PROGRAM PRG_ManualControl
VAR
	
	rMotorsActualPosition : ARRAY[1..3] OF LREAL;
	rValvesActualPosition : ARRAY[1..5] OF LREAL;
	rPumpsActualPosition  : ARRAY[1..10] OF LREAL;
	rDegreesPerVolume 	  : ARRAY[1..10] OF LREAL;
	
	aPumpsActivated		  : ARRAY[1..10] OF BOOL;
	aPumpsDirection		  : ARRAY[1..10] OF E_PumpDirection;
	aPumpsSpeed			  : ARRAY[1..10] OF REAL;
	aPumpsVolume		  : ARRAY[1..10] OF REAL;
	aPumpsDistance		  : ARRAY[1..10] OF UINT;
	bRunPumpsBySpeed	  : BOOL := FALSE;
	bRunPumpsByVolume	  : BOOL := FALSE;
	bRunPumpsByDistance	  : BOOL := FALSE;
	
	aMotorBusy	: ARRAY[1..3] OF BOOL;
	
	fbPumpsController : FB_AllPumpsController;

	i : INT; 
	
	//interlock Variables
	iTargetPosM2 : INT;
    rActualPosM3 : LREAL;
    rTol         : LREAL := 3.0; // tolerância para considerar posição "alinhada"
    bAllowMoveM2 : BOOL := TRUE;
		
END_VAR

//Motors Manual jog handling 
MotorsJog();
MotorsActualPosition();

//New Manual Screen commands test area ##########################################################
(* <Motors> -----------------------------------------------------------------------------------------------------------------------------------------------------------------------------------*)

(*<M1 Motor>*)
//Move M1 by HMI combobox manual mode
IF GVL_HMI.aManualMotorsCmd[1].bRun THEN
	GVL_HMI.aManualMotorsCmd[1].bRun := NOT GVL_Motion.aMotors[1].MoveAbsolute(	rPosition := GVL_Settings.stMachineParam.aM1Position[GVL_HMI.aManualMotorsCmd[1].iPosition],
                        														rVelocity := GVL_Settings.stMachineParam.rM1Velocity,
                        														rAcc := GVL_Settings.stMachineParam.rM1Accleration,
                       															rDec := GVL_Settings.stMachineParam.rM1Deceleration
																				);
END_IF
//Stop Moviment M1 by HMI manual mode button
IF GVL_HMI.aManualMotorsCmd[1].bStop THEN
	GVL_HMI.aManualMotorsCmd[1].bStop := NOT GVL_Motion.aMotors[1].Stop();
END_IF
(*<\M1 Motor>*)

(*<M2 Motor>*)
//Move M2 by HMI combobox manual mode
iTargetPosM2 := GVL_HMI.aManualMotorsCmd[2].iPosition;
rActualPosM3 := rMotorsActualPosition[3];

//Interlock move for M2 base on M3 position
CASE iTargetPosM2 OF
    3: // Fill Vials
        bAllowMoveM2 := (
            ABS(rActualPosM3 - GVL_Settings.stMachineParam.aM3Position[2]) <= rTol OR
            ABS(rActualPosM3 - GVL_Settings.stMachineParam.aM3Position[3]) <= rTol OR
            ABS(rActualPosM3 - GVL_Settings.stMachineParam.aM3Position[4]) <= rTol OR
            ABS(rActualPosM3 - GVL_Settings.stMachineParam.aM3Position[5]) <= rTol
        );

    4: // Calibration
        bAllowMoveM2 := ABS(rActualPosM3 - GVL_Settings.stMachineParam.aM3Position[6]) <= rTol;

    ELSE
        bAllowMoveM2 := TRUE;
END_CASE

//M2 Moviment if there is no interlock
IF GVL_HMI.aManualMotorsCmd[2].bRun THEN
    IF bAllowMoveM2 THEN
        GVL_HMI.aManualMotorsCmd[2].bRun := NOT GVL_Motion.aMotors[2].MoveAbsolute(
            rPosition := GVL_Settings.stMachineParam.aM2Position[iTargetPosM2],
            rVelocity := GVL_Settings.stMachineParam.rM2Velocity,
            rAcc := GVL_Settings.stMachineParam.rM2Accleration,
            rDec := GVL_Settings.stMachineParam.rM2Deceleration
        );
    ELSE
        GVL_HMI.aManualMotorsCmd[2].bRun := FALSE;
        // TODO: Block flag or alarm
    END_IF
END_IF

//Stop Moviment M2 by HMI manual mode button
IF GVL_HMI.aManualMotorsCmd[2].bStop THEN
	GVL_HMI.aManualMotorsCmd[2].bStop := NOT GVL_Motion.aMotors[2].Stop();
END_IF
(*<\M2 Motor>*)

(*<M3 Motor>*)
//Interlock by M2 Position
IF GVL_HMI.aManualMotorsCmd[3].bRun THEN
    IF ABS(rMotorsActualPosition[2] - GVL_Settings.stMachineParam.aM2Position[1]) > rTol THEN
        //If M2 it is not in Home Position, M3 move cannot be done
        GVL_HMI.aManualMotorsCmd[3].bRun := FALSE;
        // TODO: Block flag or alarm
    ELSE
        GVL_HMI.aManualMotorsCmd[3].bRun := NOT GVL_Motion.aMotors[3].MoveAbsolute(
            rPosition := GVL_Settings.stMachineParam.aM3Position[GVL_HMI.aManualMotorsCmd[3].iPosition],
            rVelocity := GVL_Settings.stMachineParam.rM3Velocity,
            rAcc := GVL_Settings.stMachineParam.rM3Accleration,
            rDec := GVL_Settings.stMachineParam.rM3Deceleration
        );
    END_IF
END_IF
//Stop Moviment M2 by HMI manual mode button
IF GVL_HMI.aManualMotorsCmd[3].bStop THEN
	GVL_HMI.aManualMotorsCmd[3].bStop := NOT GVL_Motion.aMotors[3].Stop();
END_IF
(*<\M3 Motor>*)

(* <Valves> -----------------------------------------------------------------------------------------------------------------------------------------------------------------------------------*)

(*<Valve 1>*)
//Move Valve 1 by HMI combobox manual mode
IF GVL_HMI.aManualValvesCmd[1].bMove THEN
	GVL_HMI.aManualValvesCmd[1].bMove := NOT GVL_Motion.aValvesObj[1].MoveValve( iPosition := GVL_HMI.aManualValvesCmd[1].iTargetPos ,rVelocity := 1500, rAcc := 1000, rDec := 1000);
END_IF

//Stop Moviment Valve 1 by HMI manual mode button
IF GVL_HMI.aManualValvesCmd[1].bStop THEN
	GVL_HMI.aManualValvesCmd[1].bStop := NOT GVL_Motion.aValvesObj[1].Stop();
END_IF
(*<\Valve 1>*)

(*<Valve 2>*)
//Move Valve 2 by HMI combobox manual mode
IF GVL_HMI.aManualValvesCmd[2].bMove THEN
	GVL_HMI.aManualValvesCmd[2].bMove := NOT GVL_Motion.aValvesObj[2].MoveValve( iPosition := GVL_HMI.aManualValvesCmd[2].iTargetPos ,rVelocity := 1500, rAcc := 1000, rDec := 1000);
END_IF

//Stop Moviment Valve 2 by HMI manual mode button
IF GVL_HMI.aManualValvesCmd[2].bStop THEN
	GVL_HMI.aManualValvesCmd[2].bStop := NOT GVL_Motion.aValvesObj[2].Stop();
END_IF
(*<\Valve 2>*)

(*<Valve 3>*)
//Move Valve 3 by HMI combobox manual mode
IF GVL_HMI.aManualValvesCmd[3].bMove THEN
	GVL_HMI.aManualValvesCmd[3].bMove := NOT GVL_Motion.aValvesObj[3].MoveValve( iPosition := GVL_HMI.aManualValvesCmd[3].iTargetPos ,rVelocity := 1500, rAcc := 1000, rDec := 1000);
END_IF

//Stop Moviment Valve 3 by HMI manual mode button
IF GVL_HMI.aManualValvesCmd[3].bStop THEN
	GVL_HMI.aManualValvesCmd[3].bStop := NOT GVL_Motion.aValvesObj[3].Stop();
END_IF
(*<\Valve 3>*)

(*<Valve 4>*)
//Move Valve 4 by HMI combobox manual mode
IF GVL_HMI.aManualValvesCmd[4].bMove THEN
	GVL_HMI.aManualValvesCmd[4].bMove := NOT GVL_Motion.aValvesObj[4].MoveValve( iPosition := GVL_HMI.aManualValvesCmd[4].iTargetPos ,rVelocity := 1500, rAcc := 1000, rDec := 1000);
END_IF

//Stop Moviment Valve 4 by HMI manual mode button
IF GVL_HMI.aManualValvesCmd[4].bStop THEN
	GVL_HMI.aManualValvesCmd[4].bStop := NOT GVL_Motion.aValvesObj[4].Stop();
END_IF
(*<\Valve 4>*)

(*<Valve 5>*)
//Move Valve 5 by HMI combobox manual mode
IF GVL_HMI.aManualValvesCmd[5].bMove THEN
	GVL_HMI.aManualValvesCmd[5].bMove := NOT GVL_Motion.aValvesObj[5].MoveValve( iPosition := GVL_HMI.aManualValvesCmd[5].iTargetPos ,rVelocity := 1500, rAcc := 1000, rDec := 1000);
END_IF

//Stop Moviment Valve 5 by HMI manual mode button
IF GVL_HMI.aManualValvesCmd[5].bStop THEN
	GVL_HMI.aManualValvesCmd[5].bStop := NOT GVL_Motion.aValvesObj[5].Stop();
END_IF
(*<\Valve 5>*)

(* <Pumps> -----------------------------------------------------------------------------------------------------------------------------------------------------------------------------------*)
(*<Move by Speed>*)
IF GVL_HMI.bRunPumpsBySpeedBt THEN //Fill up the pump arrays and trigger pumps 
	FOR i := 1 TO 10 DO
		aPumpsActivated[i] := GVL_HMI.aManualPumpsCmd[i].bActive;
		aPumpsDirection[i] := GVL_HMI.aManualPumpsCmd[i].eDirection;
		aPumpsSpeed[i] := GVL_HMI.aManualPumpsCmd[i].rSpeed * 6;
	END_FOR
	bRunPumpsBySpeed := TRUE;
	GVL_HMI.bRunPumpsBySpeedBt := FALSE;
END_IF
IF bRunPumpsBySpeed THEN //pumps movement
	bRunPumpsBySpeed := NOT fbPumpsController.MoveBySpeed(aPumpIds := aPumpsActivated, aVelocity := aPumpsSpeed, aPumpDirection := aPumpsDirection);
END_IF
(*<\Move by Speed>*)

(*<Move by Volume>*)
IF GVL_HMI.bRunPumpsByVolumeBt THEN //Fill up the pump arrays and trigger pumps 
	FOR i := 1 TO 10 DO
		aPumpsActivated[i] := GVL_HMI.aManualPumpsCmd[i].bActive;
		aPumpsDirection[i] := GVL_HMI.aManualPumpsCmd[i].eDirection;
		aPumpsSpeed[i] := GVL_HMI.aManualPumpsCmd[i].rSpeed * 6;
		aPumpsVolume[i] := GVL_HMI.aManualPumpsCmd[i].rVolume;
	END_FOR
	bRunPumpsByVolume := TRUE;
	GVL_HMI.bRunPumpsByVolumeBt := FALSE;
END_IF
IF bRunPumpsByVolume THEN //pumps movement
	bRunPumpsByVolume := NOT fbPumpsController.MoveByVolume(aPumpIds := aPumpsActivated, aVolume := aPumpsVolume, aPumpDirection := aPumpsDirection, aVelocity := aPumpsSpeed);
END_IF
(*<\Move by Volume>*)

(*<Move by Distance>*)
IF GVL_HMI.bRunPumpsByDistanceBt THEN //Fill up the pump arrays and trigger pumps 
	FOR i := 1 TO 10 DO
		aPumpsActivated[i] := GVL_HMI.aManualPumpsCmd[i].bActive;
		aPumpsDirection[i] := GVL_HMI.aManualPumpsCmd[i].eDirection;
		aPumpsSpeed[i] := GVL_HMI.aManualPumpsCmd[i].rSpeed * 6;
		aPumpsDistance[i] := GVL_HMI.aManualPumpsCmd[i].iDistance;
	END_FOR
	bRunPumpsByDistance := TRUE;
	GVL_HMI.bRunPumpsByDistanceBt := FALSE;
END_IF
IF bRunPumpsByDistance THEN //pumps movement
	bRunPumpsByDistance := NOT fbPumpsController.MoveByDistance(aPumpIds := aPumpsActivated, aRevolutions := aPumpsDistance, aPumpDirection := aPumpsDirection, aVelocity := aPumpsSpeed);
END_IF
(*<\Move by Distance>*)

(*<Stop All Pumps>*)
IF GVL_HMI.bStopPumpsBt THEN
	GVL_HMI.bStopPumpsBt := NOT fbPumpsController.StopAllPumps();
END_IF
(*<\Stop All Pumps>*)

(* <\Pumps> ----------------------------------------------------------------------------------------------------------------------------------------------------------------------------------*)

ACTION MotorsActualPosition:
// Get Motors Actual Position
rMotorsActualPosition[1] := GVL_Motion.aMotors[1].GetPosition();
rMotorsActualPosition[2] := GVL_Motion.aMotors[2].GetPosition();
rMotorsActualPosition[3] := GVL_Motion.aMotors[3].GetPosition();
rValvesActualPosition[1] := GVL_Motion.aValvesObj[1].GetPosition();
rValvesActualPosition[2] := GVL_Motion.aValvesObj[2].GetPosition();
rValvesActualPosition[3] := GVL_Motion.aValvesObj[3].GetPosition();
rValvesActualPosition[4] := GVL_Motion.aValvesObj[4].GetPosition();
rValvesActualPosition[5] := GVL_Motion.aValvesObj[5].GetPosition();
rPumpsActualPosition[1] := GVL_Motion.aPumpsLinear[1].GetPosition();
rPumpsActualPosition[2] := GVL_Motion.aPumpsLinear[2].GetPosition();
rPumpsActualPosition[3] := GVL_Motion.aPumpsLinear[3].GetPosition();
rPumpsActualPosition[4] := GVL_Motion.aPumpsLinear[4].GetPosition();
rPumpsActualPosition[5] := GVL_Motion.aPumpsLinear[5].GetPosition();
rPumpsActualPosition[6] := GVL_Motion.aPumpsLinear[6].GetPosition();
rPumpsActualPosition[7] := GVL_Motion.aPumpsLinear[7].GetPosition();
rPumpsActualPosition[8] := GVL_Motion.aPumpsLinear[8].GetPosition();
rPumpsActualPosition[9] := GVL_Motion.aPumpsLinear[9].GetPosition();
rPumpsActualPosition[10] := GVL_Motion.aPumpsLinear[10].GetPosition();

//Linear Motors - M1, M2, M3
GVL_Motion.M1Motor.rActualPosition := F_ROUND_REAL(rInput := TO_REAL(rMotorsActualPosition[1]), iDecimalPlaces := 2)* -1;
GVL_Motion.M2Motor.rActualPosition := F_ROUND_REAL(rInput := TO_REAL(rMotorsActualPosition[2]), iDecimalPlaces := 2)* -1;
GVL_Motion.M3Motor.rActualPosition := F_ROUND_REAL(rInput := TO_REAL(rMotorsActualPosition[3]), iDecimalPlaces := 2)* -1;

//Vici Valves - M4 to M8
GVL_Motion.aValves[1].rActualPosition := F_ROUND_REAL(rInput := TO_REAL(rValvesActualPosition[1]), iDecimalPlaces := 2);
GVL_Motion.aValves[2].rActualPosition := F_ROUND_REAL(rInput := TO_REAL(rValvesActualPosition[2]), iDecimalPlaces := 2);
GVL_Motion.aValves[3].rActualPosition := F_ROUND_REAL(rInput := TO_REAL(rValvesActualPosition[3]), iDecimalPlaces := 2);
GVL_Motion.aValves[4].rActualPosition := F_ROUND_REAL(rInput := TO_REAL(rValvesActualPosition[4]), iDecimalPlaces := 2);
GVL_Motion.aValves[5].rActualPosition := F_ROUND_REAL(rInput := TO_REAL(rValvesActualPosition[5]), iDecimalPlaces := 2);

//Linear pumps - 1 to 10
GVL_Motion.aPumps[1].Linear.rActualPosition  := F_ROUND_REAL(rInput := TO_REAL(rPumpsActualPosition[1]), iDecimalPlaces := 2)* -1;
GVL_Motion.aPumps[2].Linear.rActualPosition  := F_ROUND_REAL(rInput := TO_REAL(rPumpsActualPosition[2]), iDecimalPlaces := 2)* -1;
GVL_Motion.aPumps[3].Linear.rActualPosition  := F_ROUND_REAL(rInput := TO_REAL(rPumpsActualPosition[3]), iDecimalPlaces := 2)* -1;
GVL_Motion.aPumps[4].Linear.rActualPosition  := F_ROUND_REAL(rInput := TO_REAL(rPumpsActualPosition[4]), iDecimalPlaces := 2)* -1;
GVL_Motion.aPumps[5].Linear.rActualPosition  := F_ROUND_REAL(rInput := TO_REAL(rPumpsActualPosition[5]), iDecimalPlaces := 2)* -1;
GVL_Motion.aPumps[6].Linear.rActualPosition  := F_ROUND_REAL(rInput := TO_REAL(rPumpsActualPosition[6]), iDecimalPlaces := 2)* -1;
GVL_Motion.aPumps[7].Linear.rActualPosition  := F_ROUND_REAL(rInput := TO_REAL(rPumpsActualPosition[7]), iDecimalPlaces := 2)* -1;
GVL_Motion.aPumps[8].Linear.rActualPosition  := F_ROUND_REAL(rInput := TO_REAL(rPumpsActualPosition[8]), iDecimalPlaces := 2)* -1;
GVL_Motion.aPumps[9].Linear.rActualPosition  := F_ROUND_REAL(rInput := TO_REAL(rPumpsActualPosition[9]), iDecimalPlaces := 2)* -1;
GVL_Motion.aPumps[10].Linear.rActualPosition := F_ROUND_REAL(rInput := TO_REAL(rPumpsActualPosition[10]), iDecimalPlaces := 2)* -1;
END_ACTION

ACTION MotorsJog:
//Manual Motors Moviment

//Manual Moviment motor 1 - Stage Collection Vertical Axis
GVL_Motion.aMotors[1].Jog(bFwd := GVL_HMI.ManualMov.bMotorsJogFwd[1], bBwd := GVL_HMI.ManualMov.bMotorsJogBwd[1]);
//Manual Moviment motor 2 - Sample Recovery Vertical Axis
GVL_Motion.aMotors[2].Jog(bFwd := GVL_HMI.ManualMov.bMotorsJogFwd[2], bBwd := GVL_HMI.ManualMov.bMotorsJogBwd[2]);
//Manual Moviment motor 3 - Sample Recovery Horizontal Axis
GVL_Motion.aMotors[3].Jog(bFwd := GVL_HMI.ManualMov.bMotorsJogFwd[3], bBwd := GVL_HMI.ManualMov.bMotorsJogBwd[3]);

//Manual Moviment M4 - Valve 1 
GVL_Motion.aValvesObj[1].Jog(bFwd := GVL_HMI.ManualMov.bValvesJogFwd[1], bBwd := GVL_HMI.ManualMov.bValvesJogBwd[1]);
//Manual Moviment M5 - Valve 2 
GVL_Motion.aValvesObj[2].Jog(bFwd := GVL_HMI.ManualMov.bValvesJogFwd[2], bBwd := GVL_HMI.ManualMov.bValvesJogBwd[2]);
//Manual Moviment M6 - Valve 3
GVL_Motion.aValvesObj[3].Jog(bFwd := GVL_HMI.ManualMov.bValvesJogFwd[3], bBwd := GVL_HMI.ManualMov.bValvesJogBwd[3]);
//Manual Moviment M7 - Valve 4
GVL_Motion.aValvesObj[4].Jog(bFwd := GVL_HMI.ManualMov.bValvesJogFwd[4], bBwd := GVL_HMI.ManualMov.bValvesJogBwd[4]);
//Manual Moviment M8 - Valve 5
GVL_Motion.aValvesObj[5].Jog(bFwd := GVL_HMI.ManualMov.bValvesJogFwd[5], bBwd := GVL_HMI.ManualMov.bValvesJogBwd[5]);

//Manual Moviment Pump 1 - Linear
GVL_Motion.aPumpsLinear[1].Jog(bFwd := GVL_HMI.ManualMov.bPumpsLinearJogFwd[1], bBwd := GVL_HMI.ManualMov.bPumpsLinearJogBwd[1]);
//Manual Moviment Pump 2 - Linear
GVL_Motion.aPumpsLinear[2].Jog(bFwd := GVL_HMI.ManualMov.bPumpsLinearJogFwd[2], bBwd := GVL_HMI.ManualMov.bPumpsLinearJogBwd[2]);
//Manual Moviment Pump 3 - Linear
GVL_Motion.aPumpsLinear[3].Jog(bFwd := GVL_HMI.ManualMov.bPumpsLinearJogFwd[3], bBwd := GVL_HMI.ManualMov.bPumpsLinearJogBwd[3]);
//Manual Moviment Pump 4 - Linear
GVL_Motion.aPumpsLinear[4].Jog(bFwd := GVL_HMI.ManualMov.bPumpsLinearJogFwd[4], bBwd := GVL_HMI.ManualMov.bPumpsLinearJogBwd[4]);
//Manual Moviment Pump 5 - Linear
GVL_Motion.aPumpsLinear[5].Jog(bFwd := GVL_HMI.ManualMov.bPumpsLinearJogFwd[5], bBwd := GVL_HMI.ManualMov.bPumpsLinearJogBwd[5]);
//Manual Moviment Pump 6 - Linear
GVL_Motion.aPumpsLinear[6].Jog(bFwd := GVL_HMI.ManualMov.bPumpsLinearJogFwd[6], bBwd := GVL_HMI.ManualMov.bPumpsLinearJogBwd[6]);
//Manual Moviment Pump 7 - Linear
GVL_Motion.aPumpsLinear[7].Jog(bFwd := GVL_HMI.ManualMov.bPumpsLinearJogFwd[7], bBwd := GVL_HMI.ManualMov.bPumpsLinearJogBwd[7]);
//Manual Moviment Pump 8 - Linear
GVL_Motion.aPumpsLinear[8].Jog(bFwd := GVL_HMI.ManualMov.bPumpsLinearJogFwd[8], bBwd := GVL_HMI.ManualMov.bPumpsLinearJogBwd[8]);
//Manual Moviment Pump 9 - Linear
GVL_Motion.aPumpsLinear[9].Jog(bFwd := GVL_HMI.ManualMov.bPumpsLinearJogFwd[9], bBwd := GVL_HMI.ManualMov.bPumpsLinearJogBwd[9]);
//Manual Moviment Pump 10 - Linear
GVL_Motion.aPumpsLinear[10].Jog(bFwd := GVL_HMI.ManualMov.bPumpsLinearJogFwd[10], bBwd := GVL_HMI.ManualMov.bPumpsLinearJogBwd[10]);
END_ACTION

END_PROGRAM

(* stored: Version 1.1.0.1, ProductVersion 3.1.4024.15
   POU PRG_ManualControl: Id {d07ba183-6201-49c6-acdd-4e668144af08}, SpecialFunc None
   Action MotorsActualPosition: Id {634c759f-49ee-43fa-86d1-7097ca0492ea}
   Action MotorsJog: Id {57b89f50-f3a8-44a2-8323-78bd3226c039} *)
